TYPE Astrofan612FfuConfig EXTENDS DeviceConfiguration :
STRUCT
	SpeedMatrix	: FfuMatrixconfig;
	Loop : Astrofan612FfuLoopConfig;
END_STRUCT
END_TYPE

(* stored: Version 1.1.0.1, ProductVersion 3.1.4024.12
   DUT Astrofan612FfuConfig: Id {c7a64adb-b9ee-4a61-aa17-22e75e2e9b57} *)
